FUNCTION_BLOCK Zone
VAR_INPUT
END_VAR
VAR_OUTPUT
END_VAR
VAR
END_VAR

//

END_FUNCTION_BLOCK

(* stored: Version 1.1.0.1, ProductVersion 3.1.4026.8
   POU Zone: Id {555fce11-eff5-0ccb-1ed8-8a44af541b59}, SpecialFunc None *)
